INTERFACE I_Visitor

METHOD VisitElementA
VAR_INPUT
	in_fbElementA		:FB_ElementA;
END_VAR
END_METHOD

METHOD VisitElementB
VAR_INPUT
	in_fbElementB		:FB_ElementB;
END_VAR
END_METHOD

END_INTERFACE

(* stored: Version 1.1.0.1
   Itf I_Visitor: Id {8be74490-4e0b-49cb-85a9-c8f8d0afde03}
   Method VisitElementA: Id {bfbda618-9f0e-44cc-a0ba-0cd7851009e5}
   Method VisitElementB: Id {9e4d5e7c-b782-442b-823c-d6b579710ecb} *)
